60:
	ComRead(xExecute := TRUE,hCom:= com, pBuffer:= ADR(ack_buffer2), szBuffer:= SIZEOF(ack_buffer2));			
	IF ComRead.xError THEN
		atcState := 32767;
	END_IF
	IF ComRead.xDone THEN
		position := find(ack_buffer2, 'SEND OK');
		IF position > 0 THEN
			actionState := 255;
		ELSE
			actionState := 0;
		END_IF
		ComRead(xExecute := FALSE, hCom:= com);
		loop_count2 := loop_count2 + 1;
		IF loop_count2 > 50 THEN
			loop_count2 := 0;
			actionState := 32767;
		END_IF
	END_IF
	
255:
	xDone := TRUE;
	xError := FALSE;
	xBusy := FALSE;
	actionState := 250;

	loop_count1 := 0;
	loop_count2 := 0; 
	ack_buffer1 := '';
	ack_buffer2 := '';
	qisend_buffer := 'AT+QISEND=';	
	
250:

32767:
	xDone := FALSE;
	xError := TRUE;
	xBusy := FALSE;
	actionState := 32700;

	loop_count1 := 0;
	loop_count2 := 0; 
	ack_buffer1 := '';
	ack_buffer2 := '';
	qisend_buffer := 'AT+QISEND=';	
	
32700:

END_CASE

END_FUNCTION_BLOCK

// Changsha_Xiangji_ARM_Cortex_A9_xilinx_zynq7000_linux/Application/gprs_lib/UDP_Read
FUNCTION_BLOCK UDP_Read
VAR_INPUT
	xExecute:BOOL := FALSE;
	com :CAA.HANDLE;
	buffer: CAA.PVOID;
	rsize : CAA.SIZE;
END_VAR
VAR_OUTPUT
	xDone :BOOL := FALSE;
	xBusy :BOOL := FALSE;
	xError :BOOL := FALSE;
	size :CAA.SIZE;
	
END_VAR
VAR
	ton_fb :TON;  
	ComWrite: COM.Write;
	ComRead: COM.Read;	
	ack_buffer :STRING[1499];
	position :INT := -1;
	qird :STRING := 'AT+QIRD=0,1,0,1500$R';

	read_data_buffer: ARRAY[0..1499] OF BYTE;
	i :INT;
	read_num :INT;
	comma1 :INT;
	comma2 :INT;
	new_line :INT;
	data_len :INT := 0;
	//uchar *pos, *comma1, *comma2, *new_line;
	
	loop_count :INT := 0;
	
	del_atcState :INT;
	iStat :UINT := 0;
END_VAR

IF com = 0 OR NOT xExecute THEN
	xDone := FALSE;
	xError := FALSE;
	xBusy := FALSE;
	iStat := 0;
	ComRead(xExecute := FALSE);
	RETURN;
END_IF

CASE iStat OF
	0:
	ComRead(xExecute := TRUE,hCom:= com, pBuffer:= ADR(ack_buffer), szBuffer:= SIZEOF(ack_buffer));			
	IF ComRead.xError THEN
		iStat := 32767;
	END_IF
	IF ComRead.xDone THEN
		position := find(ack_buffer, '+QIRDI: 0,1,0');
		IF position > 0 THEN
			iStat := 2;
		ELSE
			iStat := 1;
		END_IF
		ComRead(xExecute := FALSE, hCom:= com);
		loop_count := loop_count + 1;
		IF loop_count > 10 THEN
			iStat := 2;
		END_IF
	END_IF
	
	1:
	ton_fb(IN := TRUE, PT := TIME#100MS);
	IF (ton_fb.Q) THEN
		ton_fb(IN := FALSE, PT := TIME#100MS);
		iStat := 0;
	END_IF
	
	2:
	ComWrite(xExecute := TRUE, hCom:= com, pBuffer:= ADR(qird), szSize:= len(qird));
	IF ComWrite.xError THEN
		iStat := 32767;
	END_IF
	
	IF ComWrite.xDone THEN
		iStat := 3;
		ComWrite(xExecute := FALSE, hCom:= com);	
	END_IF
	
	3:
	ton_fb(IN := TRUE, PT := TIME#300MS);
	IF (ton_fb.Q) THEN
		ton_fb(IN := FALSE, PT := TIME#300MS);
		iStat := 4;
	END_IF
	
	4:
	ComRead(xExecute := TRUE,hCom:= com, pBuffer:= ADR(read_data_buffer), szBuffer:= rsize);			
	IF ComRead.xError THEN
		iStat := 32767;
	END_IF
	IF ComRead.xDone THEN
		iStat := 5;
		read_num :=  ANY_TO_INT(ComRead.szSize);
		ComRead(xExecute := FALSE, hCom:= com);		
	END_IF
	
	5: //查找第一个逗号，第二次读取的时候，会返回OK，表示已经读完
	IF read_num = 6 THEN
		iStat := 255;
		RETURN;
	END_IF
	FOR i := 0 TO read_num - 1 BY 1 DO
		iStat := 32767;
		IF read_data_buffer[i] = 16#2C THEN
			comma1 := i;
			iStat := 6;
			RETURN;
		END_IF
	END_FOR;
	
	6: //查找第二个逗号
	FOR i := comma1 + 1 TO read_num - 1 BY 1 DO
		iStat := 32767;
		IF read_data_buffer[i] = 16#2C THEN
			comma2 := i;
			iStat := 7;
			RETURN;
		END_IF
	END_FOR;
	
	7: //查找回车换行
	FOR i := comma2 + 1 TO read_num - 1 BY 1 DO
		iStat := 32767;
		IF read_data_buffer[i] = 16#0D  AND read_data_buffer[i + 1] = 16#0A THEN
			new_line := i;
			iStat := 8;
			RETURN;
		END_IF
	END_FOR;
	
	8: // 获取数据长度
	FOR i := comma2 + 1 TO new_line - 1 BY 1 DO
		data_len := data_len *10 + read_data_buffer[i] - 16#30;
	END_FOR;

	iStat := 255;
	IF data_len > 0 THEN
		size := data_len;
		SysMemCpy(pDest:=buffer,pSrc:=ADR(read_data_buffer) + new_line + 2, udiCount:=data_len);
		
		data_len := 0;
		ack_buffer := '';
		loop_count := 0;
		read_num := 0;
		FOR i := 0 TO 1499 BY 1 DO
			read_data_buffer[i] := 0;
		END_FOR
		iStat := 2;
	END_IF
	
	255:
		ComRead(xExecute := FALSE);
		xDone := TRUE;
		xBusy := FALSE;
		xError := FALSE;
		iStat := 256;
		
		data_len := 0;
		ack_buffer := '';
		loop_count := 0;
		read_num := 0;
		FOR i := 0 TO 1499 BY 1 DO
			read_data_buffer[i] := 0;
		END_FOR		
	256:
	
	32767:
		ComRead(xExecute := FALSE);
		xError := TRUE;
		xDone := FALSE;
		xBusy := FALSE;
		iStat := 32700;
		
		data_len := 0;
		ack_buffer := '';
		loop_count := 0;
		read_num := 0;
		FOR i := 0 TO 1499 BY 1 DO
			read_data_buffer[i] := 0;
		END_FOR		
	32700:
	
END_CASE

END_FUNCTION_BLOCK

// Changsha_Xiangji_ARM_Cortex_A9_xilinx_zynq7000_linux/Application/GPRS/File_Read
FUNCTION_BLOCK File_Read
VAR_INPUT
	file_name :STRING;
END_VAR
VAR_OUTPUT
	sReadLine		: STRING;
	isRead          :BOOL := FALSE;	
END_VAR
VAR
	hfile			: CAA.HANDLE;
	FileOpen 		: File.Open;
	FileClose		: File.Close;
	FileRead		: File.Read;
	
	iState			: UINT := 0;	
	xError			: BOOL := FALSE;
END_VAR

 CASE iState OF
	0: // Open the file again, with read access.
	   isRead := false;
	   FileOpen(xExecute:= TRUE, sFileName:= file_name, xExclusive:= FALSE, eFileMode:= File.MODE.MREAD);
	   IF FileOpen.xDone = TRUE THEN
		   hfile := FileOpen.hFile;
		   FileOpen(xExecute:= FALSE);
		   iState := 1;
		   sReadLine := '';
	   ELSIF FileOpen.xError = TRUE THEN
		   iState:= 32767;
		   FileOpen(xExecute:= FALSE);
	   END_IF

	1: // Read the string from the file.
	   FileRead(xExecute:= TRUE, hFile:= hfile, pBuffer:= ADR(sReadLine), szBuffer:= SIZEOF(sReadLine));
	   IF FileRead.xDone = TRUE THEN
		   iState := 2;		   
		   sReadLine := MID(sReadLine, ANY_TO_INT(FileRead.szSize), 1);
		   FileRead(xExecute:= FALSE);
	   ELSIF FileRead.xError = TRUE THEN
		   iState:= 32767;
		   FileRead(xExecute:= FALSE);
	   END_IF 
	   
	 2: // Close that file.
	   FileClose(xExecute:= TRUE, hFile:= hfile);
	   IF FileClose.xDone = TRUE THEN
		   iState := 3;
		   FileClose(xExecute:= FALSE);
	   ELSIF FileClose.xError = TRUE THEN
		   iState:= 32767;
		   FileClose(xExecute:= FALSE);
	   END_IF
	   
	3: 	  
		isRead := TRUE;
		iState := 0;
		
	32767: 		
	
END_CASE

END_FUNCTION_BLOCK

// Changsha_Xiangji_ARM_Cortex_A9_xilinx_zynq7000_linux/Application/gprs_lib/Com_Read
FUNCTION_BLOCK Com_Read
VAR_INPUT
	xExecute:BOOL := FALSE;
	com :CAA.HANDLE;
	wbuffer: CAA.PVOID;
	wsize :CAA.SIZE;	
	rbuffer: CAA.PVOID;
	rsize : CAA.SIZE;
END_VAR
VAR_OUTPUT
	xDone:BOOL := FALSE;
	xBusy:BOOL := FALSE;
	xError:BOOL := FALSE;
	size :CAA.SIZE;
END_VAR
VAR
	iState :INT;
	ton_fb :TON;  
	ComWrite: COM.Write;
	ComRead: COM.Read;	
	actionState :INT;
END_VAR

IF NOT xExecute THEN
	iState := 0;
	xDone := FALSE;
	xBusy := FALSE;
	xError := FALSE;
	size := 0;
	RETURN;
END_IF

CASE iState OF
0:
	size := 0;
	ComWrite(xExecute := TRUE, hCom:= com, pBuffer:= wbuffer, szSize:= wsize);
	IF ComWrite.xError THEN
		iState := 32767;
	END_IF
	IF ComWrite.xDone THEN
		iState := 10;
		ComWrite(xExecute := FALSE, hCom:= com);	
	END_IF
	xBusy := TRUE;
	
10:
	ton_fb(IN := TRUE, PT := TIME#300MS);
	IF (ton_fb.Q) THEN
		ton_fb(IN := FALSE, PT := TIME#300MS);
		iState := 20;
	END_IF
	
20:
	ComRead(xExecute := TRUE,hCom:= com, pBuffer:= rbuffer, szBuffer:= rsize);			
	IF ComRead.xError THEN
		iState := 32767;
	END_IF
	IF ComRead.xDone THEN
		iState := 255;
		size := ComRead.szSize;
		ComRead(xExecute := FALSE, hCom:= com);		
	END_IF
	
255:
	xDone := TRUE;
	xBusy := FALSE;
	
32767:
	xError := TRUE;
	
END_CASE

END_FUNCTION_BLOCK

// Changsha_Xiangji_ARM_Cortex_A9_xilinx_zynq7000_linux/Application/GPRS/Packet_Heart
FUNCTION_BLOCK Packet_Heart
VAR_INPUT
	device_sn :STRING;
	iccd_str :STRING;
	lac_num :UINT;
	cid_num :UINT;
	worktime :UDINT;
END_VAR
VAR_OUTPUT
	heart_buffer : ARRAY[0..250] OF BYTE;
END_VAR
VAR
	heart_state :INT := 0;
	sub_str :STRING;
	num :UINT;
	packet_seq :BYTE := 0;
	iccid_code :ARRAY[0..9] OF BYTE;
	i : INT;
	
	total :UINT := 0;
	
END_VAR

//1. CMA123456781234
//1.1 CMA
heart_buffer[0] := device_sn[0];
heart_buffer[1] := device_sn[1];
heart_buffer[2] := device_sn[2];

// 1.2 12
sub_str := mid(device_sn, 2, 4);
heart_buffer[3] := STRING_TO_BYTE(sub_str);

// 1.3 34
sub_str := mid(device_sn, 2, 6);
heart_buffer[4] := STRING_TO_BYTE(sub_str);

// 1.4 56
sub_str := mid(device_sn, 2, 8);
heart_buffer[5] := STRING_TO_BYTE(sub_str);

// 1.5 78
sub_str := mid(device_sn, 2, 10);
heart_buffer[6] := STRING_TO_BYTE(sub_str);

// 1.6 1234
sub_str := mid(device_sn, 4, 12);
num := STRING_TO_UINT(sub_str);
heart_buffer[7] := ANY_TO_BYTE(num / 256);
heart_buffer[8] := ANY_TO_BYTE(num MOD 256);

// 2. protocol version
heart_buffer[9] := 0;

// 3. data length
heart_buffer[10] := 0;
heart_buffer[11] := 81;

// 4. data type
heart_buffer[12] := 16#01;

// 5. data seq
heart_buffer[13] := packet_seq;
packet_seq := packet_seq + 1;

// 6. parameter
heart_buffer[14] := 0;

// 7. version
heart_buffer[15] := 0;

// 8. reserved 1
heart_buffer[16] := 0;

// 9. reserved 2
heart_buffer[17] := 0;

// 10. length
heart_buffer[18] := 0;
heart_buffer[19] := 73;

// 11. LAC 
heart_buffer[20] := ANY_TO_BYTE(lac_num / 256);
heart_buffer[21] := ANY_TO_BYTE(lac_num MOD 256);

// 12. CID 
heart_buffer[22] := ANY_TO_BYTE(cid_num / 256);
heart_buffer[23] := ANY_TO_BYTE(cid_num MOD 256);

// 13. iccid
iccid_code := Iccid_Get(iccd_str);
FOR i := 0 TO 9 DO
	heart_buffer[24 + i] := iccid_code[i];
END_FOR

// 14. work time
heart_buffer[34] := ANY_TO_BYTE(worktime / 65536 /256);
heart_buffer[35] := ANY_TO_BYTE(worktime / 65536 MOD 256);
heart_buffer[36] := ANY_TO_BYTE(worktime MOD 65536 / 256);
heart_buffer[37] := ANY_TO_BYTE(worktime MOD 65536 MOD 256);

// 15. customer code
heart_buffer[38] := 0;
heart_buffer[39] := 0;

// 16. local host code
heart_buffer[40] := 0;
heart_buffer[41] := 0;

//**********以下为GPRS回传数据**************//
heart_buffer[42].0 := FALSE;
heart_buffer[42].1 := FALSE;
heart_buffer[42].2 := FALSE;
heart_buffer[42].3 := FALSE;
heart_buffer[42].4 := FALSE;
heart_buffer[42].5 := FALSE;
heart_buffer[42].6 := FALSE;
heart_buffer[42].7 := FALSE;

heart_buffer[43].0 := FALSE;
heart_buffer[43].1 := Wastewater_full_Fault;//污水满故障
heart_buffer[43].2 := T_DI_oil_filter_block.Q;//回油过滤堵塞
heart_buffer[43].3 := T_DI_oil_level_low.Q;//液压油位低故障
heart_buffer[43].4 := FALSE;
heart_buffer[43].5 := T_DI_cleanwater_LOW.Q;//水箱缺水故障
heart_buffer[43].6 := FALSE;
heart_buffer[43].7 := DI_Rcar_fault;//倒车故障停机

heart_buffer[44].0 := Wastewater_full_Fault1;//污水满故障停机
heart_buffer[44].1 := NOT DI_power_on;//电源故障
heart_buffer[44].2 := T_Pumpspeed_H.Q;//高压水泵超速报警
heart_buffer[44].3 := T_Pumpspeed_HH.Q;//高压水泵超速停止
heart_buffer[44].4 := TEST_ALM;//请关闭测试
heart_buffer[44].5 := RCAR_ALM;//正在倒车中提示
heart_buffer[44].6 := Motor_Work_ALM;//请先启动电机提示
heart_buffer[44].7 := Func_test_HMI;//测试打开

heart_buffer[45].0 := T_DI_air_press_low.Q;//气路系统压力低
heart_buffer[45].1 := T_DI_Rcar.Q;//倒车
heart_buffer[45].2 := FALSE;
heart_buffer[45].3 := DO_Hpre_pump_noWork;//高压水泵未啮合
heart_buffer[45].4 := T_Chassis_SOC_LOW.Q;//底盘电量低停机
heart_buffer[45].5 := DI_Hpre_valve_noOpen;//高压吹净球阀未打开
heart_buffer[45].6 := DI_Totvalve_noOpen;//高压水路球阀未打开
heart_buffer[45].7 := DO_Box_Up_arm;//请先打开箱门

heart_buffer[46].0 := fog_Spump_arm;//隔膜泵球阀未打开
heart_buffer[46].1 := T_fog_pump_press_noOk.Q;//隔膜泵压力不正常
heart_buffer[46].2 := Fault_STOP;//故障停机
heart_buffer[46].3 := DO_Box_Down_arm;//请先放下撑杆
heart_buffer[46].4 := T_DI_wastewater_full.Q;//主污水箱水满
heart_buffer[46].5 := Backup_power_Test_warn;//请先打开备用动力开关
heart_buffer[46].6 := T_Chassis_CAN_fault.Q;//底盘CAN通讯故障
heart_buffer[46].7 := T_Motor_CAN_fault.Q;//与电机CAN通讯故障

heart_buffer[47].0 := T_auxiliary_warte_dif.Q;//辅污水箱水位不一致
heart_buffer[47].1 := T_DI_auxiliary1_warte_H.Q;//辅1污水箱水满
heart_buffer[47].2 := T_DI_auxiliary2_warte_H.Q;//辅2污水箱水满
heart_buffer[47].3 := T_water_overflow_noClose.Q;//水路卸荷阀未关闭故障
heart_buffer[47].4 := T_water_overflow_noOpen.Q;//水路卸荷阀未打开故障
heart_buffer[47].5 := DI_backup_power_open;//备用动力打开提示
heart_buffer[47].6 := Chassis_SOC_LOW;//底盘电量低压20%提示
heart_buffer[47].7 := High_voltage_noReady;//底盘未上高压提示

heart_buffer[48].0 := (DI_cleanwater_LOW<3000);
heart_buffer[48].1 := DI_Totvalve_Open;
heart_buffer[48].2 := DI_box_door_close;
heart_buffer[48].3 := DI_Hpre_valve_open;
heart_buffer[48].4 := DI_air_press_low;
heart_buffer[48].5 := DI_wastewater_full;
heart_buffer[48].6 := DI_Rod_noDown;
heart_buffer[48].7 := DI_backup_power_open;

heart_buffer[49].0 := DI_water_overflow;
heart_buffer[49].1 := FALSE;
heart_buffer[49].2 := FALSE;
heart_buffer[49].3 := FALSE;
heart_buffer[49].4 := DI_fog_pump_press_ok;
heart_buffer[49].5 := DI_oil_level_low;
heart_buffer[49].6 := DI_oil_filter_block;
heart_buffer[49].7 := FALSE;

heart_buffer[50].0 := DI_power_on;
heart_buffer[50].1 := DI_Rcar;
heart_buffer[50].2 := DI_oil_release_valve;
heart_buffer[50].3 := FALSE;
heart_buffer[50].4 := DI_auxiliary1_warte_H;
heart_buffer[50].5 := DI_auxiliary2_warte_H;
heart_buffer[50].6 := DI_Sweep_Up;
heart_buffer[50].7 := DI_Sweep_Down;

heart_buffer[51].0 := DI_sweep_out;
heart_buffer[51].1 := DI_sweep_return;
heart_buffer[51].2 := FALSE;
heart_buffer[51].3 := FALSE;
heart_buffer[51].4 := FALSE;
heart_buffer[51].5 := FALSE;
heart_buffer[51].6 := FALSE;
heart_buffer[51].7 := FALSE;

heart_buffer[52].0 := DO_Lsweep_down;
heart_buffer[52].1 := DO_Lsweep_up;
heart_buffer[52].2 := DO_Rsweep_down;
heart_buffer[52].3 := DO_Rsweep_up;
heart_buffer[52].4 := DO_Lsweep_out;
heart_buffer[52].5 := DO_Rsweep_out;
heart_buffer[52].6 := DO_Lrod_out;
heart_buffer[52].7 := DO_Rrod_out;

heart_buffer[53].0 := DO_pointshoot_up;
heart_buffer[53].1 := DO_pointshoot_down;
heart_buffer[53].2 := DO_pointshoot_left;
heart_buffer[53].3 := DO_pointshoot_right;
heart_buffer[53].4 := FALSE;
heart_buffer[53].5 := DO_water_overflow;
heart_buffer[53].6 := DO_Lrod_water;
heart_buffer[53].7 := DO_Rrod_water;

heart_buffer[54].0 := DO_Suction_water;
heart_buffer[54].1 := DO_Hpressure_water;
heart_buffer[54].2 := DO_selfclean_water;
heart_buffer[54].3 := DO_Hpre_pump;
heart_buffer[54].4 := DO_fog_Spump;
heart_buffer[54].5 := DO_Motor_en;
heart_buffer[54].6 := DO_watercooler_pump;
heart_buffer[54].7 := DO_cooler_fan;

heart_buffer[55].0 := DO_backup_power;
heart_buffer[55].1 := DO_wastewater_valve;
heart_buffer[55].2 := DO_wastewater_pump;
heart_buffer[55].3 := DO_oil_release_valve;
heart_buffer[55].4 := DO_Sweep_Mspeed;
heart_buffer[55].5 := DO_Sweep_Lspeed;
heart_buffer[55].6 := DO_RSweep;
heart_buffer[55].7 := DO_LASweep;

heart_buffer[56].0 := DO_RASweep;
heart_buffer[56].1 := DO_Box_Down;
heart_buffer[56].2 := DO_Box_Up;
heart_buffer[56].3 := DO_Suction_Down;
heart_buffer[56].4 := DO_Suction_Up;
heart_buffer[56].5 := DO_Door_Open;
heart_buffer[56].6 := DO_Door_Close;
heart_buffer[56].7 := FALSE;

heart_buffer[57].0 := FALSE;
heart_buffer[57].1 := FALSE;
heart_buffer[57].2 := FALSE;
heart_buffer[57].3 := FALSE;
heart_buffer[57].4 := FALSE;
heart_buffer[57].5 := FALSE;
heart_buffer[57].6 := FALSE;
heart_buffer[57].7 := FALSE;

heart_buffer[58].0 := AwashSweep_HMI;
heart_buffer[58].1 := LwashSweep_HMI;
heart_buffer[58].2 := RwashSweep_HMI;
heart_buffer[58].3 := ASweeproad_HMI;
heart_buffer[58].4 := LSweeproad_HMI;
heart_buffer[58].5 := RSweeproad_HMI;
heart_buffer[58].6 := Aclean_HMI;
heart_buffer[58].7 := Lclean_HMI;

heart_buffer[59].0 := Rclean_HMI;
heart_buffer[59].1 := Sweep_stop_HMI;
heart_buffer[59].2 := DO_fog_Spump1;
heart_buffer[59].3 := DO_selfclean_water1;
heart_buffer[59].4 := DO_Door_Close1;
heart_buffer[59].5 := DO_Door_Open1;
heart_buffer[59].6 := DO_Box_Up1;
heart_buffer[59].7 := DO_Box_Down1;

heart_buffer[60].0 := FALSE;
heart_buffer[60].1 := FALSE;
heart_buffer[60].2 := FALSE;
heart_buffer[60].3 := FALSE;
heart_buffer[60].4 := Standard_speed_HMI;
heart_buffer[60].5 := Strong_speed_HMI;
heart_buffer[60].6 := Sweep_HSpeed_HMI;
heart_buffer[60].7 := Sweep_MSpeed_HMI;

heart_buffer[61].0 := Sweep_LSpeed_HMI;
heart_buffer[61].1 := DO_Hpressure_water1;
heart_buffer[61].2 := Drain_start_HMI;
heart_buffer[61].3 := Drain_auto_HMI;
heart_buffer[61].4 := Drain_manual_HMI;
heart_buffer[61].5 := Lrod_drain_HMI;
heart_buffer[61].6 := Rrod_drain_HMI;
heart_buffer[61].7 := Hpressure_drain_HMI;

heart_buffer[62].0 := Selfclean_drain_HMI;
heart_buffer[62].1 := replace_Sweep_HMI;
heart_buffer[62].2 := Func_test_HMI;
heart_buffer[62].3 := Intelligent_HMI;
heart_buffer[62].4 := Cleanly_HMI;
heart_buffer[62].5 := Normal_HMI;
heart_buffer[62].6 := Dirty_HMI;
heart_buffer[62].7 := DO_wastewater_pump_open1;

heart_buffer[63].0 := Pointshoot_up_HMI;
heart_buffer[63].1 := Pointshoot_down_HMI;
heart_buffer[63].2 := Pointshoot_left_HMI;
heart_buffer[63].3 := Pointshoot_right_HMI;
heart_buffer[63].4 := Suction_drain_HMI;
heart_buffer[63].5 := FALSE;
heart_buffer[63].6 := motor_work;
heart_buffer[63].7 := sys_work;

heart_buffer[64] := ANY_TO_BYTE(Motor_real_torque_HMI MOD 256);
heart_buffer[65] :=ANY_TO_BYTE(Motor_real_torque_HMI/256);

heart_buffer[66] :=ANY_TO_BYTE(Motor_real_speed_HMI MOD 256);
heart_buffer[67] :=ANY_TO_BYTE(Motor_real_speed_HMI/256);

heart_buffer[68] :=ANY_TO_BYTE(Motor_bus_voltage_HMI MOD 256);
heart_buffer[69] :=ANY_TO_BYTE(Motor_bus_voltage_HMI/256);

heart_buffer[70] :=ANY_TO_BYTE(Motor_phase_current_HMI MOD 256);
heart_buffer[71] :=ANY_TO_BYTE(Motor_phase_current_HMI/256);

heart_buffer[72] :=ANY_TO_BYTE(Motor_max_dirve_torque_HMI MOD 256);
heart_buffer[73] :=ANY_TO_BYTE(Motor_max_dirve_torque_HMI/256);

heart_buffer[74] :=ANY_TO_BYTE(Motor_max_brake_torque_HMI MOD 256);
heart_buffer[75] :=ANY_TO_BYTE(Motor_max_brake_torque_HMI/256);

heart_buffer[76] :=Motor_temp_controller_HMI;
heart_buffer[77] :=Motor_temp_HMI;

heart_buffer[78] :=ANY_TO_BYTE(Motor_max_speed_HMI MOD 256);
heart_buffer[79] :=ANY_TO_BYTE(Motor_max_speed_HMI/256);

heart_buffer[80] := 0*1+Motor_direction_cw*4+Motor_mode*16+Motor_stat*64;
heart_buffer[81] := Motor_bus_low_voltage*1+Motor_bus_high_voltage*4+MOtor_ctrller_high_temp*16+Motor_high_temp*64;
heart_buffer[82] := Motor_igbt_fault*1+Motor_overspeed*4+Motor_comm_error*16+Motor_short*64;
heart_buffer[83] := Motor_overload*1+Motor_selfcheck_fault*4+Motor_low_voltage*16+Motor_sensor_fault*64;

heart_buffer[84] := Chassis_Soc;//底盘电量

heart_buffer[85] :=ANY_TO_BYTE(16#201 MOD 256);
heart_buffer[86] :=ANY_TO_BYTE(16#201/256);

heart_buffer[87] :=ANY_TO_BYTE(Chassis_speed MOD 256);
heart_buffer[88] :=ANY_TO_BYTE(Chassis_speed/256);//底盘车速

heart_buffer[89] :=ANY_TO_BYTE(motor_work_time MOD 256);
heart_buffer[90] :=ANY_TO_BYTE(motor_work_time/16#100);
heart_buffer[91] :=ANY_TO_BYTE(motor_work_time/16#10000);
heart_buffer[92] :=ANY_TO_BYTE(motor_work_time/16#1000000);


//**********以上为GPRS回传数据**************//

//以下为校验需要放到最后
total := 0;
FOR i := 0 TO 92 DO    (* 90代表GPRS回传的数据字节总数 *)
	total := total + heart_buffer[i];
END_FOR

// 15. taotal check
heart_buffer[93] := ANY_TO_BYTE(total / 256);
heart_buffer[94] := ANY_TO_BYTE(total MOD 256);

END_FUNCTION_BLOCK

// Changsha_Xiangji_ARM_Cortex_A9_xilinx_zynq7000_linux/Application/GPRS/fb_get_iccid
FUNCTION_BLOCK fb_get_iccid
VAR_INPUT
	xExecute:BOOL := FALSE;
	m26_handle:CAA.HANDLE; 
END_VAR

VAR_OUTPUT
	iccid:STRING(32);
	xDone:BOOL := FALSE;
	xBusy :BOOL := FALSE;
	xError:BOOL := FALSE;
END_VAR

VAR
	iStat:UINT := 0;
	udp_handle :CAA.HANDLE; 
	accid_cmd :STRING := 'AT+ICCID$r';
	iccid_read_buffer :STRING(255);
	com_read :Com_Read;
	udp_init_fb: INT;
	size:CAA.SIZE;
	position :INT := -1;
	ICCID_HEAD:STRING := '+ICCID: ';
END_VAR


IF NOT xExecute OR m26_handle = 0 THEN
	xDone := FALSE;
	xBusy := FALSE;
	xError := FALSE;
	iccid := '';
	RETURN;
END_IF 		

IF iccid <> '' THEN  //已经读到了，不需再读
	xDone := TRUE;
	xBusy := FALSE;
	xError := FALSE;
	RETURN; 
END_IF

CASE iStat OF
0:
	com_read(xExecute := FALSE);
	iStat := 10;
	com_read.xExecute := TRUE;
10:
	IF com_read.xDone THEN
		IF com_read.size > 0 THEN
			position := find(iccid_read_buffer, ICCID_HEAD);
			IF position > 0 THEN
				iccid := mid(iccid_read_buffer, 20, position + len(ICCID_HEAD));
				xDone := TRUE;
				iStat := 100;
			END_IF
		END_IF
	ELSIF com_read.xError THEN
		xDone := FALSE;
		iStat := 200;
	END_IF	
100:

200:

END_CASE

com_read(com:= m26_handle, wbuffer:= ADR(accid_cmd), wsize := len(accid_cmd), rbuffer := ADR(iccid_read_buffer), rsize := SIZEOF(iccid_read_buffer));

END_FUNCTION_BLOCK

// Changsha_Xiangji_ARM_Cortex_A9_xilinx_zynq7000_linux/Application/GPRS/fb_get_lac
FUNCTION_BLOCK fb_get_lac
VAR_INPUT
	xExecute:BOOL := FALSE;
	m26_handle:CAA.HANDLE; 
END_VAR
VAR_OUTPUT
	lac:STRING(4) := '0000';
	ci :STRING(4) := '0000';
	xDone:BOOL := FALSE;
	xError:BOOL := FALSE;
END_VAR
VAR
	iStat:UINT := 0;
	udp_handle :CAA.HANDLE; 
	lac_set_cmd :STRING := 'AT+CREG=2$r';
	lac_get_cmd :STRING := 'AT+CREG?$r';
	lac_close_cmd :STRING := 'AT+CREG=0$r';
	lac_read_buffer :STRING(255);
	com_read :Com_Read;
	udp_init_fb: INT;
	size:CAA.SIZE;
	position :INT := -1;
	LACID_HEAD:STRING := '+CREG:';
	lac_str:STRING(8);
	ci_str:STRING(8);
END_VAR


IF m26_handle = 0 THEN
	RETURN;
END_IF

IF NOT xExecute THEN
	xDone := FALSE;
	xError := FALSE;
	lac := '0000';
	ci := '0000';
	iStat := 0;
	
	RETURN;
END_IF 		

CASE iStat OF
0:
	com_read(xExecute := FALSE);
	com_read.wbuffer:= ADR(lac_set_cmd);
 	com_read.wsize := len(lac_set_cmd);
	com_read.xExecute := TRUE;	
	iStat := 5;
5:  //set m26 for lac and ci with command:  AT+CREG=2
	IF com_read.xDone THEN
		size := com_read.size;
		IF size > 0 THEN
			position := find(lac_read_buffer, 'OK');
			IF position > 0 THEN
				com_read(xExecute := FALSE);
				com_read.wbuffer:= ADR(lac_get_cmd);
				com_read.wsize := len(lac_get_cmd);
				com_read.xExecute := TRUE;				
				iStat := 10;
			END_IF
		END_IF
	ELSIF com_read.xError THEN
		xDone := FALSE;
	END_IF	

10:  //read lac and ci with command: AT+CREG?
	IF com_read.xDone THEN
		IF com_read.size > 0 THEN
			position := find(lac_read_buffer, LACID_HEAD);
			IF position > 0 THEN
				position := find(lac_read_buffer, '$"');
				IF position > 0 THEN
					lac := mid(lac_read_buffer, 4, position + 1);
					ci := mid(lac_read_buffer, 4, position + 8);
					iStat := 20;
					com_read(xExecute := FALSE);
					com_read.wbuffer:= ADR(lac_close_cmd);
 					com_read.wsize := len(lac_close_cmd);
					com_read.xExecute := TRUE;
				END_IF
			ELSE
				iStat := 0;
			END_IF
		END_IF
	ELSIF com_read.xError THEN
		xDone := FALSE;
	END_IF	
	
20:  //close
	IF com_read.xDone THEN
		size := com_read.size;
		IF size > 0 THEN
			position := find(lac_read_buffer, 'OK');
			IF position > 0 THEN
				iStat := 100;
				xDone := TRUE;
			END_IF
		END_IF
	ELSIF com_read.xError THEN
		xDone := FALSE;
	END_IF	
100: //ok

END_CASE

com_read(com:= m26_handle, rbuffer := ADR(lac_read_buffer), rsize := SIZEOF(lac_read_buffer));

END_FUNCTION_BLOCK

// Changsha_Xiangji_ARM_Cortex_A9_xilinx_zynq7000_linux/Application/GPRS/fb_m26
FUNCTION_BLOCK fb_m26
VAR_INPUT
	enable :BOOL := FALSE;
	ipaddr :STRING(32);
	port :UINT;
END_VAR
VAR_OUTPUT
	xBusy :BOOL := FALSE;
	xError :BOOL := FALSE;
	handle_m26 :CAA.HANDLE; 
END_VAR
VAR
	udp_init:Udp_Init;
	iStat :UINT := 0;
END_VAR

IF NOT enable THEN
	xBusy := FALSE;
	xError := FALSE;
	handle_m26 := 0;
	RETURN;
END_IF

CASE iStat OF
0:
	udp_init(xExecute := FALSE, ip_addr := ipaddr, port := port);
	udp_init.xExecute := TRUE;
	iStat := 10;
	
10:
	IF udp_init.xDone THEN
		xBusy := TRUE;
		handle_m26 := udp_init.udp_handle;
		iStat := 100;
	ELSIF udp_init.xError THEN
		iStat := 200;
	END_IF	

100:

200:

END_CASE


udp_init(ip_addr := ipaddr, port := port);

END_FUNCTION_BLOCK

// Changsha_Xiangji_ARM_Cortex_A9_xilinx_zynq7000_linux/Application/funcs/is_hex
FUNCTION is_hex : bool
VAR_INPUT
	ch:STRING(1);
END_VAR
VAR
END_VAR

is_hex := FALSE;
IF (ch >= '0' AND ch <= '9') OR (ch >= 'a' AND ch <= 'f') OR (ch >= 'A' AND ch <= 'F') THEN
	is_hex := TRUE;
END_IF 

RETURN;

END_FUNCTION

// Changsha_Xiangji_ARM_Cortex_A9_xilinx_zynq7000_linux/Application/main
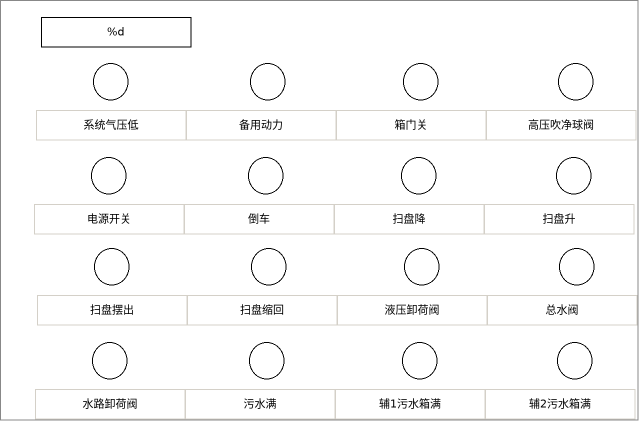
VISUALIZATION main  // 639x421
    RoundedRectangle (41,17 150x30), "%d", text variable: Motor_real_speed_HMI
    Ellipse (93,63 35x37), colour toggle: DI_air_press_low
    Textfield (36,110 150x30), "系统气压低"
    Ellipse (250,63 35x37), colour toggle: DI_backup_power_open
    Textfield (186,110 150x30), "备用动力"
    Ellipse (403,63 35x37), colour toggle: DI_box_door_close
    Textfield (336,110 150x30), "箱门关"
    Ellipse (558,63 35x37), colour toggle: DI_Hpre_valve_open
    Textfield (486,110 150x30), "高压吹净球阀"
    Ellipse (91,157 35x37), colour toggle: DI_power_on
    Textfield (34,204 150x30), "电源开关"
    Ellipse (248,157 35x37), colour toggle: DI_Rcar
    Textfield (184,204 150x30), "倒车"
    Ellipse (401,157 35x37), colour toggle: DI_Sweep_Down
    Textfield (334,204 150x30), "扫盘降"
    Ellipse (556,157 35x37), colour toggle: DI_Sweep_Up
    Textfield (484,204 150x30), "扫盘升"
    Ellipse (94,248 35x37), colour toggle: DI_sweep_out
    Textfield (37,295 150x30), "扫盘摆出"
    Ellipse (251,248 35x37), colour toggle: DI_sweep_return
    Textfield (187,295 150x30), "扫盘缩回"
    Ellipse (404,248 35x37), colour toggle: DI_oil_release_valve
    Textfield (337,295 150x30), "液压卸荷阀"
    Ellipse (559,248 35x37), colour toggle: DI_Totvalve_Open
    Textfield (487,295 150x30), "总水阀"
    Ellipse (92,342 35x37), colour toggle: DI_water_overflow
    Textfield (35,389 150x30), "水路卸荷阀"
    Ellipse (249,342 35x37), colour toggle: DI_wastewater_full
    Textfield (185,389 150x30), "污水满"
    Ellipse (402,342 35x37), colour toggle: DI_auxiliary1_warte_H
    Textfield (335,389 150x30), "辅1污水箱满"
    Ellipse (557,342 35x37), colour toggle: DI_auxiliary2_warte_H
    Textfield (485,389 150x30), "辅2污水箱满"
END_VISUALIZATION
